// TIA Portal V16 export
// export: Created 2023-06-21T17:06:29.4132913Z, ExportSetting WithDefaults, DisplayName Totally Integrated Automation Portal, DisplayVersion V16 Update 4, DisplayName TIA Portal Version Control Interface, DisplayVersion V16 Update 2, DisplayName TIA Portal Openness, DisplayVersion V16 Update 4, DisplayName SINAMICS Startdrive Advanced, DisplayVersion V16, DisplayName SINAMICS Startdrive G130, G150, S120, S150, SINAMICS MV, S210, DisplayVersion V16, DisplayName SINAMICS Startdrive G110M, G120, G120C, G120D, G120P, DisplayVersion V16, DisplayName STEP 7 Professional, DisplayVersion V16 Update 4, DisplayName STEP 7 Safety, DisplayVersion V16, DisplayName Soft Starter ES, DisplayVersion V16, DisplayName WinCC Advanced, DisplayVersion V16 Update 4
VAR_GLOBAL   // PLC tag table "Default tag table"
   System_Byte AT %MB1 : Byte;
   FirstScan AT %M1.0 : Bool;
   DiagStatusUpdate AT %M1.1 : Bool;
   AlwaysTRUE AT %M1.2 : Bool;
   AlwaysFALSE AT %M1.3 : Bool;
   Clock_Byte AT %MB0 : Byte;
   Clock_10Hz AT %M0.0 : Bool;
   Clock_5Hz AT %M0.1 : Bool;
   "Clock_2.5Hz" AT %M0.2 : Bool;
   Clock_2Hz AT %M0.3 : Bool;
   "Clock_1.25Hz" AT %M0.4 : Bool;
   Clock_1Hz AT %M0.5 : Bool;
   "Clock_0.625Hz" AT %M0.6 : Bool;
   "Clock_0.5Hz" AT %M0.7 : Bool;
   Aux_1 AT %M2.0 : Bool;
   START_COMM AT %M2.1 : Bool;
   BS_03 AT %M2.6 : Bool;
   Comm_ok AT %M2.3 : Bool;
   Count_Modbus AT %MW50 : Word;
   RST_Count AT %M49.0 : Bool;
   Tag_2 AT %M49.1 : Bool;
   Tag_3 AT %M49.2 : Bool;
   Tag_4 AT %M49.3 : Bool;
   Tag_5 AT %M49.4 : Bool;
   MB_DONE_COUNT AT %MW54 : Word;
   Tag_7 AT %M49.7 : Bool;
   MB_ERROR_COUNT AT %MW58 : Word;
   MB_STATUS AT %MW62 : Word;
   Tag_10 AT %M30.0 : Bool;
   Tag_11 AT %MW70 : Word;
   Tag_12 AT %MW74 : Word;
   Tag_13 AT %MW78 : Word;
   Liga_01 AT %M3.0 : Bool;
   Desliga_01 AT %M3.1 : Bool;
   Liga_02 AT %M3.2 : Bool;
   Desliga_02 AT %M3.3 : Bool;
   Liga_03 AT %M3.4 : Bool;
   Desliga_03 AT %M3.5 : Bool;
   Liga_04 AT %M3.6 : Bool;
   Desliga_04 AT %M3.7 : Bool;
   Liga_05 AT %M4.0 : Bool;
   Desliga_05 AT %M4.1 : Bool;
   Liga_06 AT %M4.2 : Bool;
   Desliga_06 AT %M4.3 : Bool;
   Liga_07 AT %M4.4 : Bool;
   Desliga_07 AT %M4.5 : Bool;
   Liga_08 AT %M4.6 : Bool;
   Desliga_08 AT %M4.7 : Bool;
   Liga_09 AT %M5.0 : Bool;
   Desliga_09 AT %M5.1 : Bool;
   Liga_10 AT %M5.2 : Bool;
   Desliga_10 AT %M5.3 : Bool;
   Liga_11 AT %M5.4 : Bool;
   Desliga_11 AT %M5.5 : Bool;
   Liga_12 AT %M5.6 : Bool;
   Desliga_12 AT %M5.7 : Bool;
   Liga_13 AT %M6.0 : Bool;
   Desliga_13 AT %M6.1 : Bool;
   Liga_14 AT %M6.2 : Bool;
   Desliga_14 AT %M6.3 : Bool;
   Oper_Mode_01 AT %MW80 : Word;
   SP_01 AT %MW82 : Word;
   Oper_Mode_02 AT %MW84 : Word;
   SP_02 AT %MW86 : Word;
   Oper_Mode_03 AT %MW88 : Word;
   SP_03 AT %MW90 : Word;
   Oper_Mode_04 AT %MW92 : Word;
   SP_04 AT %MW94 : Word;
   Oper_Mode_05 AT %MW96 : Word;
   SP_05 AT %MW98 : Word;
   Oper_Mode_06 AT %MW100 : Word;
   SP_06 AT %MW102 : Word;
   Oper_Mode_07 AT %MW104 : Word;
   SP_07 AT %MW106 : Word;
   Oper_Mode_08 AT %MW108 : Word;
   SP_08 AT %MW110 : Word;
   Oper_Mode_09 AT %MW112 : Word;
   SP_09 AT %MW114 : Word;
   Oper_Mode_10 AT %MW116 : Word;
   SP_10 AT %MW118 : Word;
   Oper_Mode_11 AT %MW120 : Word;
   SP_11 AT %MW122 : Word;
   Oper_Mode_12 AT %MW124 : Word;
   SP_12 AT %MW126 : Word;
   Oper_Mode_13 AT %MW128 : Word;
   SP_13 AT %MW130 : Word;
   Oper_Mode_14 AT %MW132 : Word;
   SP_14 AT %MW134 : Word;
   Tag_1 AT %M7.1 : Bool;
   Timeout_Desligado_Counter AT %M6.4 : Bool;
   Timeout_Ligado_Counter AT %M6.5 : Bool;
   Tag_8 AT %M6.6 : Bool;
   Tag_6 AT %M6.7 : Bool;
   MB_CT_DONE AT %M7.2 : Bool;
   MB_CT_ERROR AT %M7.3 : Bool;
   Sts_Auto AT %M7.4 : Bool;
   Tag_9 AT %MW240 : Word;
   Tag_14 AT %MD242 : Real;
   "1" AT %MD246 : Real;
   Tag_15 AT %MW242 : Word;
END_VAR
